// Mitsubishi GX Works2 project: pr2   PLC: Q03UDV

PROGRAM MAIN
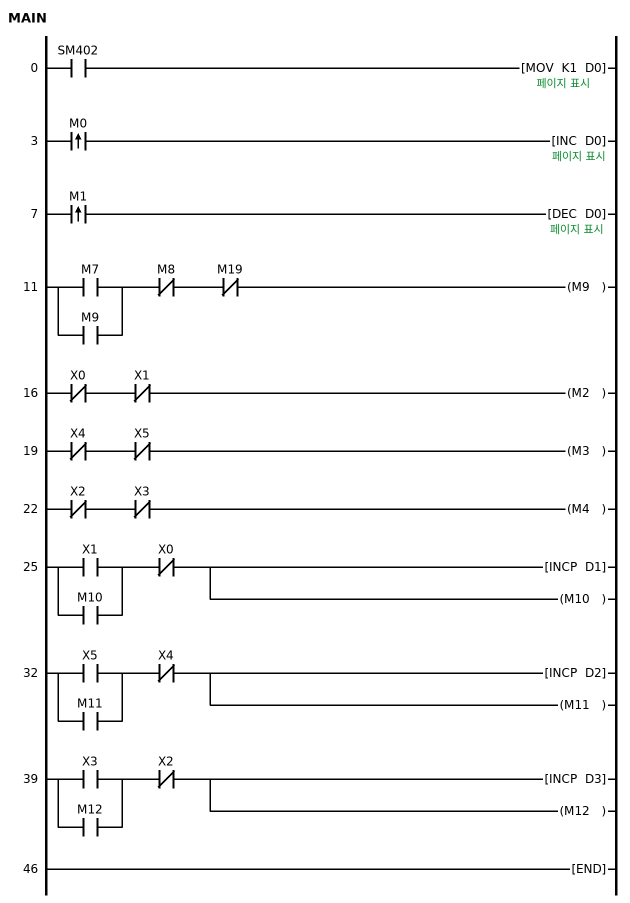
0     LD      SM402
      MOV     K1 D0  ; 페이지 표시
3     LDP     M0
      INC     D0
7     LDP     M1
      DEC     D0
11    LD      M7
      OR      M9
      ANI     M8
      ANI     M19
      OUT     M9
16    LDI     X0
      ANI     X1
      OUT     M2
19    LDI     X4
      ANI     X5
      OUT     M3
22    LDI     X2
      ANI     X3
      OUT     M4
25    LD      X1
      OR      M10
      ANI     X0
      INCP    D1
      OUT     M10
32    LD      X5
      OR      M11
      ANI     X4
      INCP    D2
      OUT     M11
39    LD      X3
      OR      M12
      ANI     X2
      INCP    D3
      OUT     M12
46    END
END_PROGRAM

PROGRAM OUTPUT
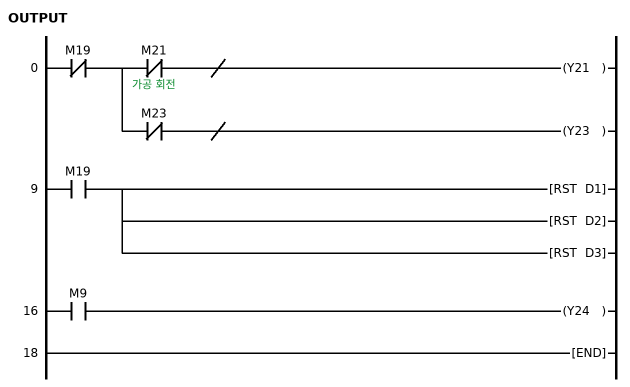
0     LDI     M19
      MPS
      ANI     M21  ; 가공 회전
      INV
      OUT     Y21
      MPP
      ANI     M23
      INV
      OUT     Y23
9     LD      M19
      RST     D1
      RST     D2
      RST     D3
16    LD      M9
      OUT     Y24
18    END
END_PROGRAM

// device comments not shown above
X15  ; 회전
X16  ; 회전 정지
X20  ; 가 모 버
X21  ; 컨 모 버
X22  ; 공 전 버
X30  ; 컨 모 버
X40  ; 공 전 버
X41  ; 공 후 버
Y0D  ; 드릴
Y2D  ; 드릴
Y2E  ; 컨베이어
M20  ; 초기화
M30  ; 컨베이어 모드
M31  ; 컨베이어 작동
